(* PLC project Tc2_System.GETCURTASKINDEX Demo, tc3-libraries-kb TwinCAT 3.1 *)
(* stored: creationDateTime 2026-05-20T00:00:00, modificationDateTime 2026-05-20T00:00:00 *)

PROGRAM P_Demo_GETCURTASKINDEX
  VAR
    fbGETCURTASKINDEX : GETCURTASKINDEX;  (* GETCURTASKINDEX 实例 *)
    nCurrentTaskIndex : BYTE;  (* 当前任务索引 1..4；FB_init 中调用结果不可靠 *)
  END_VAR

// ============================================================
// Tc2_System.GETCURTASKINDEX 演示程序
// ============================================================
// 场景：老项目里日志染色：每条日志带上任务索引便于排查。
// 价值：保留兼容旧代码；新代码改用 GETCURTASKINDEXEX 函数。
// 验证：把本 PROGRAM 加到第 2 个 PLC 任务，登录后 nCurrentTaskIndex 应为 2。
// 验证步骤：
//   1. 右键 PLC 项目 → Import PLCopenXML → 选本文件
//   2. 引用 Tc2_System（References → Add library）
//   3. 编译 → 登录 → 运行；按上方『验证』指引在线写值观察
// ============================================================

fbGETCURTASKINDEX(index => nCurrentTaskIndex);
END_PROGRAM
